TEXTLIST nEventType
  0 = ''
  1 = 'Alarm' | Deutsch: 'Alarm' | English: 'Alarm' | Turkish: 'Alarm'
  2 = 'Uyari' | Deutsch: 'Warnung' | English: 'Warning' | Turkish: 'Uyari'
  3 = 'Axis Hata'
  4 = 'NCI Hata'
  5 = 'Guvenlik'
  6 = 'SYS_Err'
   = ''
END_TEXTLIST

(* stored: Version 1.1.0.1, ProductVersion 3.1.4024.6
   TextList nEventType: Id {b75d6279-1f67-4768-9a1a-56269a2e5175} *)
